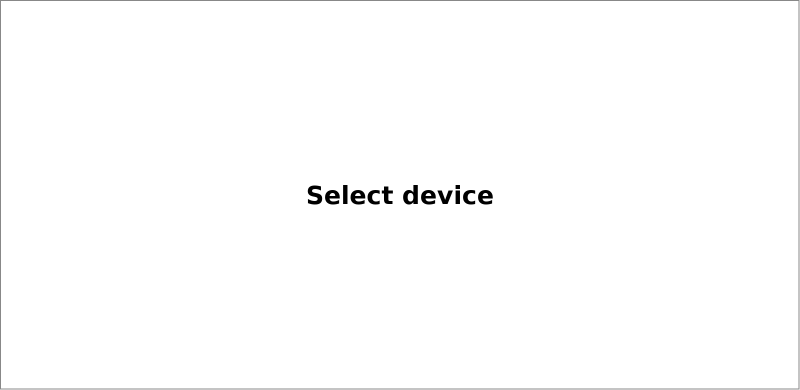
VISUALIZATION VisuUndefinedControl  // 800x390
    Label (0,0 800x390), "Select device"
END_VISUALIZATION

(* stored: Version 1.1.0.1, ProductVersion 3.1.4024.9
   Visu VisuUndefinedControl: Id {8b54ee27-69c8-402f-b826-f326a4699098} *)
